# EPICS autosave request: BPMApp/Db/AFCMgmt_settings.req
$(P)$(R)AFCSi57xFreq
$(P)$(R)AFCSi57xOe
